// TIA Portal project "FB_zad2" (V15.1)

(* hardware
DEVICE "S7-1200 station_1"  S7-1200 Station
   slot 0: "Rack_0"  S7-1200 Rack  Rack  V1.0
   slot 1: "PLC_1"  CPU 1215C DC/DC/DC  6ES7 215-1AG40-0XB0  V4.2
*)

// ===== PLC "PLC_1"  CPU 1215C DC/DC/DC =====

VAR_GLOBAL   // PLC tag table "Default tag table"
   "OS1" AT %I1.0 : Bool;
   "OS2" AT %I0.7 : Bool;
   "P1" AT %Q1.0 : Bool;
   "P2" AT %Q0.7 : Bool;
   "P3_k_stolu" AT %Q0.5 : Bool;
   "P3_k_dopravniku" AT %Q0.6 : Bool;
   "P1_pracuje" AT %M10.0 : Bool;
   "P2_pracuje" AT %M10.1 : Bool;
   "P3_pracuje" AT %M10.2 : Bool;
   "Rotating_Table" AT %Q0.4 : Bool;
   "KS1" AT %I0.3 : Bool;
   "KS2" AT %I0.6 : Bool;
   "Table_Is_Ok" AT %M10.3 : Bool;
   "D1" AT %Q0.2 : Bool;
   "OS3" AT %I0.2 : Bool;
   "kompressor" AT %Q0.0 : Bool;
   "poz2_pom" AT %M10.4 : Bool;
END_VAR

DATA_BLOCK "P1_DB"   // DB1
{ S7_Optimized_Access := 'TRUE' }
VERSION : 0.1
// stored: InstanceOfName Piston_FB
"Piston_FB"
BEGIN
   i_Sensor_Low := true;
   i_Sensor_High := true;
END_DATA_BLOCK

DATA_BLOCK "P2_DB"   // DB2
{ S7_Optimized_Access := 'TRUE' }
VERSION : 0.1
// stored: InstanceOfName Piston_FB
"Piston_FB"
BEGIN
END_DATA_BLOCK

DATA_BLOCK "P3_DB"   // DB3
{ S7_Optimized_Access := 'TRUE' }
VERSION : 0.1
// stored: InstanceOfName Piston_FB
"Piston_FB"
BEGIN
   i_Is_Big_Piston := true;
END_DATA_BLOCK

DATA_BLOCK "Table1_DB"   // DB4
{ S7_Optimized_Access := 'TRUE' }
VERSION : 0.1
// stored: InstanceOfName Rotating_Table_FB
"Rotating_Table_FB"
BEGIN
END_DATA_BLOCK

DATA_BLOCK "Conv_DB"   // DB5
{ S7_Optimized_Access := 'TRUE' }
VERSION : 0.1
// stored: InstanceOfName Conveyor_FB
"Conveyor_FB"
BEGIN
END_DATA_BLOCK

FUNCTION_BLOCK "Piston_FB"   // FB1, LAD
{ S7_Optimized_Access := 'TRUE' }
VERSION : 0.1
   VAR_INPUT
      i_Enable : Bool;   // Personal control
      i_Is_Big_Piston : Bool;   // (поршни с двумя outputs, то есть как Р3)
      i_Use_Sensors : Bool;   // (true only for P1)
      i_Sensor_Low : Bool;   // (OS1)
      i_Sensor_High : Bool;   // (OS2)
      i_Set_Count : Int;   // (N iterations)
   END_VAR
   VAR_OUTPUT
      q_Forward : Bool;   // (k stolu)
      q_Backward : Bool;   // (od stola)
      q_Done : Bool;   // (Don't work)
      q_Busy : Bool;   // (In process)
      q_Object_ID : Int;
   END_VAR
   VAR
      Timer_For_Detection : TON_TIME;
      S_Vyska_Zistena : Bool;
      Timer_Work : TON_TIME;
      Timer_Return : TON_TIME;
      s_Counter_Val : Int;
      s_Edge_Mem : Bool;
      Timer_To_Push : TON_TIME;
   END_VAR
   VAR_TEMP   // added for the SCL form of the ladder/FBD networks
      _w1 : Bool;
   END_VAR
BEGIN

REGION Network 1: Určenie výšky objektu (funguje len pre prvý piest)
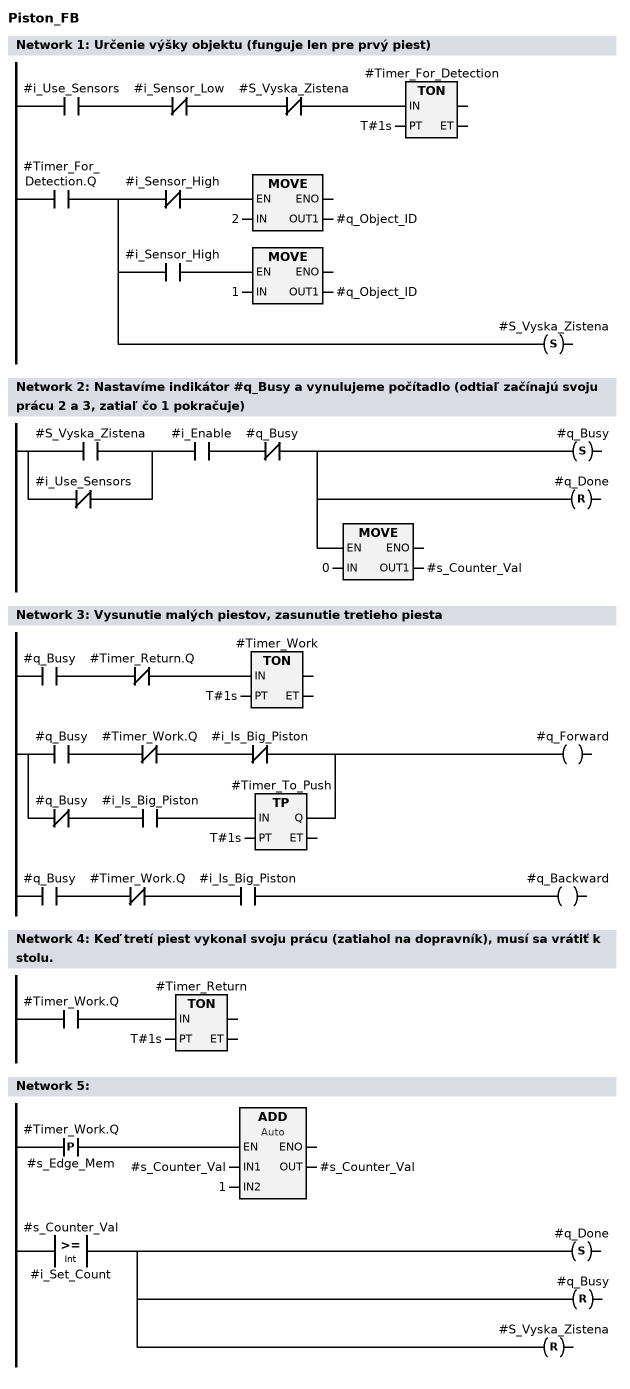
   #Timer_For_Detection(IN := #i_Use_Sensors AND NOT #i_Sensor_Low AND NOT #S_Vyska_Zistena, PT := T#1s);   // TON
   IF #Timer_For_Detection.Q AND NOT #i_Sensor_High THEN #q_Object_ID := 2; END_IF;
   IF #Timer_For_Detection.Q AND #i_Sensor_High THEN #q_Object_ID := 1; END_IF;
   IF #Timer_For_Detection.Q THEN #S_Vyska_Zistena := TRUE; END_IF;
END_REGION

REGION Network 2: Nastavíme indikátor #q_Busy a vynulujeme počítadlo (odtiaľ začínajú svoju prácu 2 a 3, zatiaľ čo 1 pokračuje)
   RUNG wire#powerrail
      Contact( #S_Vyska_Zistena )
      wire#w1
      Contact( #i_Enable )
      I_Contact( #q_Busy )
      wire#w2
      S_Coil( #q_Busy )
   END_RUNG
   RUNG wire#powerrail
      I_Contact( #i_Use_Sensors )
   END_RUNG wire#w1
   RUNG wire#w2
      R_Coil( #q_Done )
   END_RUNG
   RUNG wire#w2
      Move(in := 0, out1 => #s_Counter_Val)
   END_RUNG
   // the same network as SCL:
   #_w1 := (#S_Vyska_Zistena OR NOT #i_Use_Sensors) AND #i_Enable AND NOT #q_Busy;
   IF #_w1 THEN
       #q_Busy := TRUE;
       #q_Done := FALSE;
       #s_Counter_Val := 0;
   END_IF;
END_REGION

REGION Network 3: Vysunutie malých piestov, zasunutie tretieho piesta
   #Timer_Work(IN := #q_Busy AND NOT #Timer_Return.Q, PT := T#1s);   // TON
   #Timer_To_Push(IN := NOT #q_Busy AND #i_Is_Big_Piston, PT := T#1s);   // TP
   #q_Forward := (#q_Busy AND NOT #Timer_Work.Q AND NOT #i_Is_Big_Piston) OR #Timer_To_Push.Q;
   #q_Backward := #q_Busy AND NOT #Timer_Work.Q AND #i_Is_Big_Piston;
END_REGION

REGION Network 4: Keď tretí piest vykonal svoju prácu (zatiahol na dopravník), musí sa vrátiť k stolu.
   #Timer_Return(IN := #Timer_Work.Q, PT := T#1s);   // TON
END_REGION

REGION Network 5
   RUNG wire#powerrail
      P_Contact(operand := #Timer_Work.Q, bit := #s_Edge_Mem)
      Add(in1 := #s_Counter_Val, in2 := 1, out => #s_Counter_Val)
   END_RUNG
   RUNG wire#powerrail
      { S7_Templates := "SrcType := Int" } GE_Contact(in1 := #s_Counter_Val, in2 := #i_Set_Count)
      wire#w1
      S_Coil( #q_Done )
   END_RUNG
   RUNG wire#w1
      R_Coil( #q_Busy )
   END_RUNG
   RUNG wire#w1
      R_Coil( #S_Vyska_Zistena )
   END_RUNG
   // the same network as SCL:
   #_w1 := #Timer_Work.Q AND NOT #s_Edge_Mem;   // rising edge of #Timer_Work.Q
   #s_Edge_Mem := #Timer_Work.Q;
   IF #_w1 THEN #s_Counter_Val := #s_Counter_Val + 1; END_IF;
   IF #s_Counter_Val >= #i_Set_Count THEN
       #q_Done := TRUE;
       #q_Busy := FALSE;
       #S_Vyska_Zistena := FALSE;
   END_IF;
END_REGION
END_FUNCTION_BLOCK

FUNCTION_BLOCK "Rotating_Table_FB"   // FB2, LAD
{ S7_Optimized_Access := 'TRUE' }
VERSION : 0.1
   VAR_INPUT
      i_Enable_Auto : Bool;
      i_Enable_Manual : Bool;   // KS1
      i_Loading : Bool;   // Signal "Done" from P1_DB
      i_New_ID : Int;   // ID from P1_DB for poz1
      i_Confirm_Button : Bool;   // KS2
      i_Unloading : Bool;
   END_VAR
   VAR_OUTPUT
      q_State_Ok : Bool;
      q_Motor : Bool;
      q_Start_Poz_State : Bool;
   END_VAR
   VAR
      s_Poz1 : Int;
      s_poz2_id : Bool;
      s_Poz2 : Int;
      s_Poz3 : Int;
      s_Poz4 : Int;
      s_Block_Rotation : Bool;
      s_Need_Rotation : Bool;
      s_Rotation_Time : TON_TIME;
      s_Loading_Pom : Bool;
      s_Timer_Rotation_Pom : Bool;
      s_Timer_Rotation_Pom2 : Bool;
      s_Unloading_Pom : Bool;
      s_Rotation_Time2 : TON_TIME;
   END_VAR
   VAR_TEMP   // added for the SCL form of the ladder/FBD networks
      _w1 : Bool;
      _w2 : Bool;
   END_VAR
BEGIN

REGION Network 1
   // Vynulovanie poz3
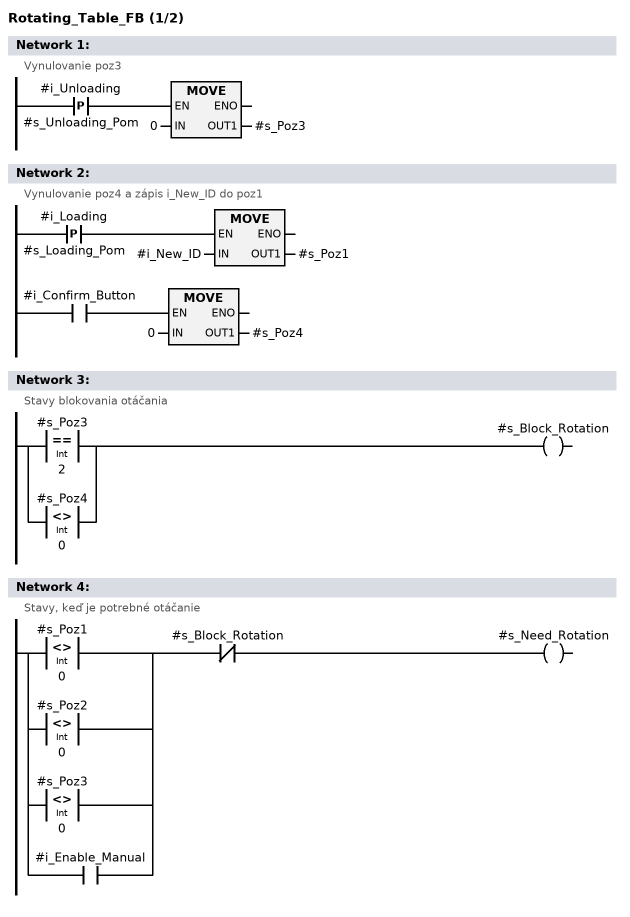
   RUNG wire#powerrail
      P_Contact(operand := #i_Unloading, bit := #s_Unloading_Pom)
      Move(in := 0, out1 => #s_Poz3)
   END_RUNG
   // the same network as SCL:
   #_w1 := #i_Unloading AND NOT #s_Unloading_Pom;   // rising edge of #i_Unloading
   #s_Unloading_Pom := #i_Unloading;
   IF #_w1 THEN #s_Poz3 := 0; END_IF;
END_REGION

REGION Network 2
   // Vynulovanie poz4 a zápis i_New_ID do poz1
   RUNG wire#powerrail
      P_Contact(operand := #i_Loading, bit := #s_Loading_Pom)
      Move(in := #i_New_ID, out1 => #s_Poz1)
   END_RUNG
   RUNG wire#powerrail
      Contact( #i_Confirm_Button )
      Move(in := 0, out1 => #s_Poz4)
   END_RUNG
   // the same network as SCL:
   #_w1 := #i_Loading AND NOT #s_Loading_Pom;   // rising edge of #i_Loading
   #s_Loading_Pom := #i_Loading;
   IF #_w1 THEN #s_Poz1 := #i_New_ID; END_IF;
   IF #i_Confirm_Button THEN #s_Poz4 := 0; END_IF;
END_REGION

REGION Network 3
   // Stavy blokovania otáčania
   RUNG wire#powerrail
      { S7_Templates := "SrcType := Int" } EQ_Contact(in1 := #s_Poz3, in2 := 2)
      wire#w1
      Coil( #s_Block_Rotation )
   END_RUNG
   RUNG wire#powerrail
      { S7_Templates := "SrcType := Int" } NE_Contact(in1 := #s_Poz4, in2 := 0)
   END_RUNG wire#w1
   // the same network as SCL:
   #s_Block_Rotation := (#s_Poz3 = 2) OR (#s_Poz4 <> 0);
END_REGION

REGION Network 4
   // Stavy, keď je potrebné otáčanie
   RUNG wire#powerrail
      { S7_Templates := "SrcType := Int" } NE_Contact(in1 := #s_Poz1, in2 := 0)
      wire#w1
      I_Contact( #s_Block_Rotation )
      Coil( #s_Need_Rotation )
   END_RUNG
   RUNG wire#powerrail
      { S7_Templates := "SrcType := Int" } NE_Contact(in1 := #s_Poz2, in2 := 0)
   END_RUNG wire#w1
   RUNG wire#powerrail
      { S7_Templates := "SrcType := Int" } NE_Contact(in1 := #s_Poz3, in2 := 0)
   END_RUNG wire#w1
   RUNG wire#powerrail
      Contact( #i_Enable_Manual )
   END_RUNG wire#w1
   // the same network as SCL:
   #s_Need_Rotation := ((#s_Poz1 <> 0) OR (#s_Poz2 <> 0) OR (#s_Poz3 <> 0) OR #i_Enable_Manual) AND NOT #s_Block_Rotation;
END_REGION

REGION Network 5
   // Určite pridanie druhého časovača (TR) nie je najstručnejším riešením, ale funguje to :))
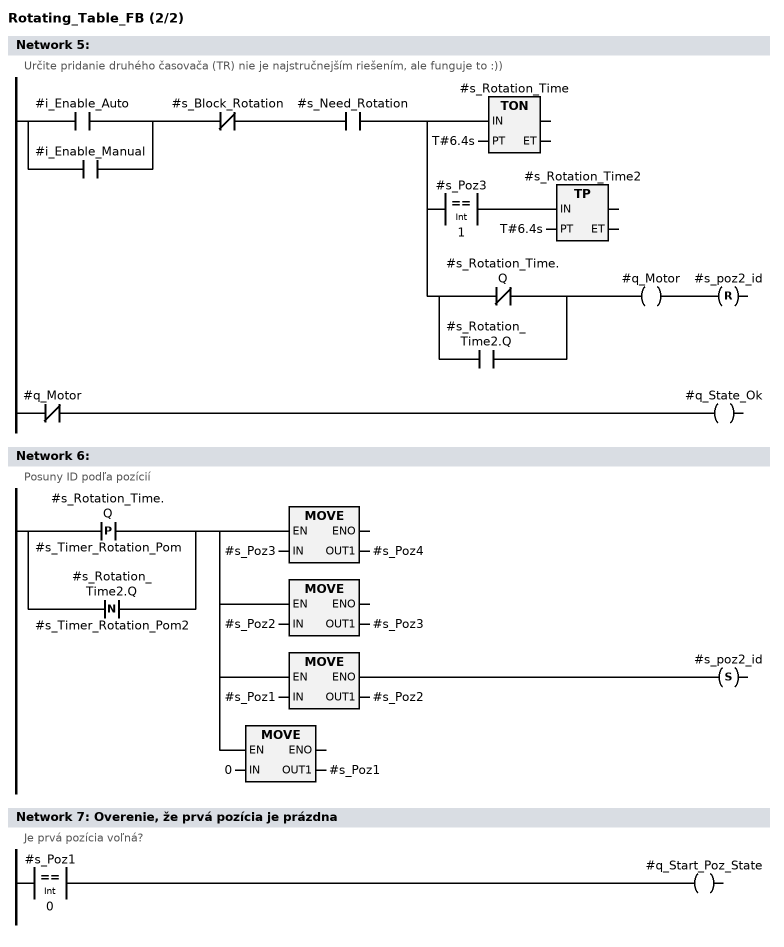
   #_w1 := (#i_Enable_Auto OR #i_Enable_Manual) AND NOT #s_Block_Rotation AND #s_Need_Rotation;
   #s_Rotation_Time(IN := #_w1, PT := T#6.4s);   // TON
   #s_Rotation_Time2(IN := #_w1 AND (#s_Poz3 = 1), PT := T#6.4s);   // TP
   #q_Motor := #_w1 AND (NOT #s_Rotation_Time.Q OR #s_Rotation_Time2.Q);
   IF #q_Motor THEN #s_poz2_id := FALSE; END_IF;
   #q_State_Ok := NOT #q_Motor;
END_REGION

REGION Network 6
   // Posuny ID podľa pozícií
   RUNG wire#powerrail
      P_Contact(operand := #s_Rotation_Time.Q, bit := #s_Timer_Rotation_Pom)
      wire#w1
      Move(in := #s_Poz3, out1 => #s_Poz4)
   END_RUNG
   RUNG wire#powerrail
      N_Contact(operand := #s_Rotation_Time2.Q, bit := #s_Timer_Rotation_Pom2)
   END_RUNG wire#w1
   RUNG wire#w1
      Move(in := #s_Poz2, out1 => #s_Poz3)
   END_RUNG
   RUNG wire#w1
      Move(in := #s_Poz1, out1 => #s_Poz2)
      S_Coil( #s_poz2_id )
   END_RUNG
   RUNG wire#w1
      Move(in := 0, out1 => #s_Poz1)
   END_RUNG
   // the same network as SCL:
   #_w1 := #s_Rotation_Time.Q AND NOT #s_Timer_Rotation_Pom;   // rising edge of #s_Rotation_Time.Q
   #s_Timer_Rotation_Pom := #s_Rotation_Time.Q;
   #_w2 := NOT #s_Rotation_Time2.Q AND #s_Timer_Rotation_Pom2;   // falling edge of #s_Rotation_Time2.Q
   #s_Timer_Rotation_Pom2 := #s_Rotation_Time2.Q;
   IF #_w1 OR #_w2 THEN
       #s_Poz4 := #s_Poz3;
       #s_Poz3 := #s_Poz2;
       #s_Poz2 := #s_Poz1;
       #s_poz2_id := TRUE;
       #s_Poz1 := 0;
   END_IF;
END_REGION

REGION Network 7: Overenie, že prvá pozícia je prázdna
   // Je prvá pozícia voľná?
   RUNG wire#powerrail
      { S7_Templates := "SrcType := Int" } EQ_Contact(in1 := #s_Poz1, in2 := 0)
      Coil( #q_Start_Poz_State )
   END_RUNG
   // the same network as SCL:
   #q_Start_Poz_State := #s_Poz1 = 0;
END_REGION
END_FUNCTION_BLOCK

FUNCTION_BLOCK "Conveyor_FB"   // FB4, LAD
{ S7_Optimized_Access := 'TRUE' }
VERSION : 0.1
   VAR_INPUT
      i_Sensor : Bool;
      i_Loading : Bool;   // Signal P3.Done
      i_New_ID : Int;
   END_VAR
   VAR_OUTPUT
      q_Motor : Bool;
      q_Entry_Is_Free : Bool;
   END_VAR
   VAR
      s_Poz5 : Int;
      s_Poz6 : Int;
      s_Is_poz6_Free : Bool;
      s_Sensor_Fall : Bool;
      s_Sensor_Rise : Bool;
      s_Loading_Pom : Bool;
   END_VAR
   VAR_TEMP   // added for the SCL form of the ladder/FBD networks
      _w1 : Bool;
   END_VAR
BEGIN

REGION Network 1: Keď piest pretiahol objekt, zapíš ID do piatej pozície
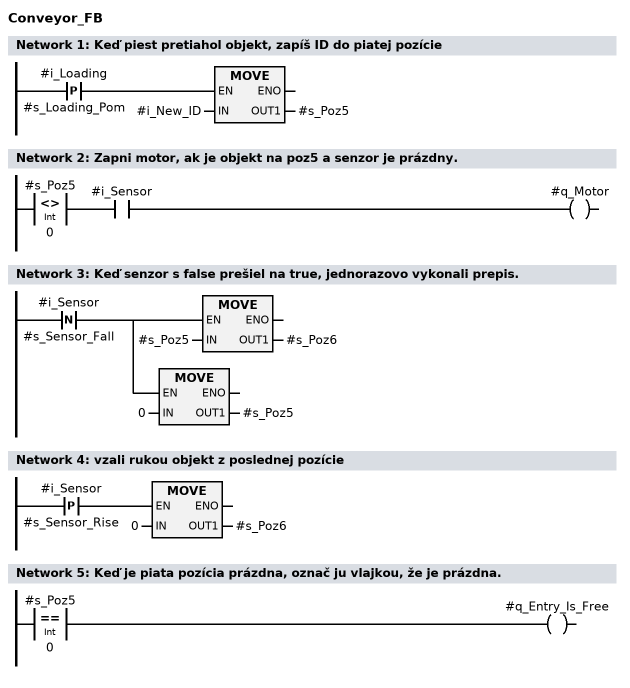
   RUNG wire#powerrail
      P_Contact(operand := #i_Loading, bit := #s_Loading_Pom)
      Move(in := #i_New_ID, out1 => #s_Poz5)
   END_RUNG
   // the same network as SCL:
   #_w1 := #i_Loading AND NOT #s_Loading_Pom;   // rising edge of #i_Loading
   #s_Loading_Pom := #i_Loading;
   IF #_w1 THEN #s_Poz5 := #i_New_ID; END_IF;
END_REGION

REGION Network 2: Zapni motor, ak je objekt na poz5 a senzor je prázdny.
   RUNG wire#powerrail
      { S7_Templates := "SrcType := Int" } NE_Contact(in1 := #s_Poz5, in2 := 0)
      Contact( #i_Sensor )
      Coil( #q_Motor )
   END_RUNG
   // the same network as SCL:
   #q_Motor := (#s_Poz5 <> 0) AND #i_Sensor;
END_REGION

REGION Network 3: Keď senzor s false prešiel na true, jednorazovo vykonali prepis.
   RUNG wire#powerrail
      N_Contact(operand := #i_Sensor, bit := #s_Sensor_Fall)
      wire#w1
      Move(in := #s_Poz5, out1 => #s_Poz6)
   END_RUNG
   RUNG wire#w1
      Move(in := 0, out1 => #s_Poz5)
   END_RUNG
   // the same network as SCL:
   #_w1 := NOT #i_Sensor AND #s_Sensor_Fall;   // falling edge of #i_Sensor
   #s_Sensor_Fall := #i_Sensor;
   IF #_w1 THEN
       #s_Poz6 := #s_Poz5;
       #s_Poz5 := 0;
   END_IF;
END_REGION

REGION Network 4: vzali rukou objekt z poslednej pozície
   RUNG wire#powerrail
      P_Contact(operand := #i_Sensor, bit := #s_Sensor_Rise)
      Move(in := 0, out1 => #s_Poz6)
   END_RUNG
   // the same network as SCL:
   #_w1 := #i_Sensor AND NOT #s_Sensor_Rise;   // rising edge of #i_Sensor
   #s_Sensor_Rise := #i_Sensor;
   IF #_w1 THEN #s_Poz6 := 0; END_IF;
END_REGION

REGION Network 5: Keď je piata pozícia prázdna, označ ju vlajkou, že je prázdna.
   RUNG wire#powerrail
      { S7_Templates := "SrcType := Int" } EQ_Contact(in1 := #s_Poz5, in2 := 0)
      Coil( #q_Entry_Is_Free )
   END_RUNG
   // the same network as SCL:
   #q_Entry_Is_Free := #s_Poz5 = 0;
END_REGION
END_FUNCTION_BLOCK

ORGANIZATION_BLOCK "Main"   // OB1, LAD, ProgramCycle
TITLE = "Main Program Sweep (Cycle)"
{ S7_Optimized_Access := 'TRUE' }
VERSION : 0.1
   VAR_INPUT
      Initial_Call : Bool;   // Initial call of this OB
      Remanence : Bool;   // =True, if remanent data are available
   END_VAR
   VAR_TEMP   // added for the SCL form of the ladder/FBD networks
      _w1 : Bool;
   END_VAR
BEGIN

REGION Network 1: Je mozno dat ( ) namiesto Set
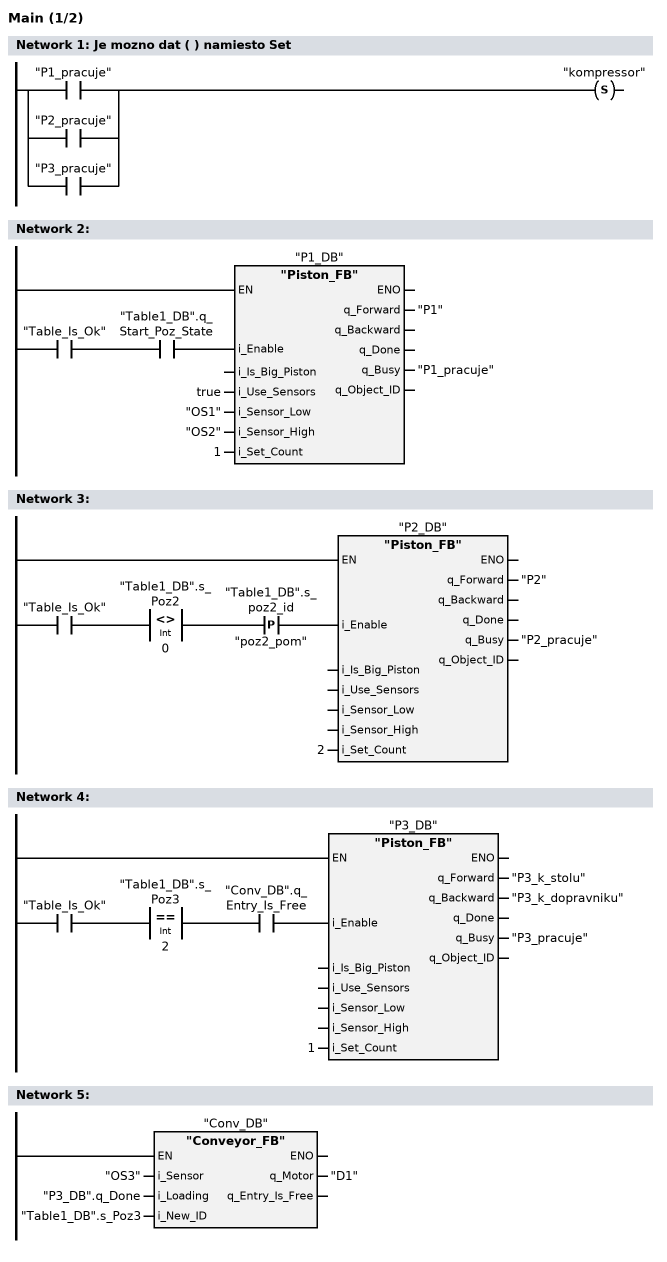
   RUNG wire#powerrail
      Contact( "P1_pracuje" )
      wire#w1
      S_Coil( "kompressor" )
   END_RUNG
   RUNG wire#powerrail
      Contact( "P2_pracuje" )
   END_RUNG wire#w1
   RUNG wire#powerrail
      Contact( "P3_pracuje" )
   END_RUNG wire#w1
   // the same network as SCL:
   IF "P1_pracuje" OR "P2_pracuje" OR "P3_pracuje" THEN "kompressor" := TRUE; END_IF;
END_REGION

REGION Network 2
   RUNG wire#powerrail
      "P1_DB"(i_Enable := wire#w1, i_Is_Big_Piston :=, i_Use_Sensors := true, i_Sensor_Low := "OS1", i_Sensor_High := "OS2", i_Set_Count := 1, q_Forward => "P1", q_Backward =>, q_Done =>, q_Busy => "P1_pracuje", q_Object_ID =>)
   END_RUNG
   RUNG wire#powerrail
      Contact( "Table_Is_Ok" )
      Contact( "Table1_DB".q_Start_Poz_State )
   END_RUNG wire#w1
   // the same network as SCL:
   "P1_DB"(i_Enable := "Table_Is_Ok" AND "Table1_DB".q_Start_Poz_State,   // "Piston_FB"
           i_Use_Sensors := true,
           i_Sensor_Low := "OS1",
           i_Sensor_High := "OS2",
           i_Set_Count := 1,
           q_Forward => "P1",
           q_Busy => "P1_pracuje");
END_REGION

REGION Network 3
   RUNG wire#powerrail
      "P2_DB"(i_Enable := wire#w1, i_Is_Big_Piston :=, i_Use_Sensors :=, i_Sensor_Low :=, i_Sensor_High :=, i_Set_Count := 2, q_Forward => "P2", q_Backward =>, q_Done =>, q_Busy => "P2_pracuje", q_Object_ID =>)
   END_RUNG
   RUNG wire#powerrail
      Contact( "Table_Is_Ok" )
      { S7_Templates := "SrcType := Int" } NE_Contact(in1 := "Table1_DB".s_Poz2, in2 := 0)
      P_Contact(operand := "Table1_DB".s_poz2_id, bit := "poz2_pom")
   END_RUNG wire#w1
   // the same network as SCL:
   #_w1 := "Table_Is_Ok" AND ("Table1_DB".s_Poz2 <> 0) AND "Table1_DB".s_poz2_id AND NOT "poz2_pom";   // rising edge of "Table1_DB".s_poz2_id
   "poz2_pom" := "Table1_DB".s_poz2_id;
   "P2_DB"(i_Enable := #_w1, i_Set_Count := 2, q_Forward => "P2", q_Busy => "P2_pracuje");   // "Piston_FB"
END_REGION

REGION Network 4
   RUNG wire#powerrail
      "P3_DB"(i_Enable := wire#w1, i_Is_Big_Piston :=, i_Use_Sensors :=, i_Sensor_Low :=, i_Sensor_High :=, i_Set_Count := 1, q_Forward => "P3_k_stolu", q_Backward => "P3_k_dopravniku", q_Done =>, q_Busy => "P3_pracuje", q_Object_ID =>)
   END_RUNG
   RUNG wire#powerrail
      Contact( "Table_Is_Ok" )
      { S7_Templates := "SrcType := Int" } EQ_Contact(in1 := "Table1_DB".s_Poz3, in2 := 2)
      Contact( "Conv_DB".q_Entry_Is_Free )
   END_RUNG wire#w1
   // the same network as SCL:
   "P3_DB"(i_Enable := "Table_Is_Ok" AND ("Table1_DB".s_Poz3 = 2) AND "Conv_DB".q_Entry_Is_Free,   // "Piston_FB"
           i_Set_Count := 1,
           q_Forward => "P3_k_stolu",
           q_Backward => "P3_k_dopravniku",
           q_Busy => "P3_pracuje");
END_REGION

REGION Network 5
   RUNG wire#powerrail
      "Conv_DB"(i_Sensor := "OS3", i_Loading := "P3_DB".q_Done, i_New_ID := "Table1_DB".s_Poz3, q_Motor => "D1", q_Entry_Is_Free =>)
   END_RUNG
   // the same network as SCL:
   "Conv_DB"(i_Sensor := "OS3", i_Loading := "P3_DB".q_Done, i_New_ID := "Table1_DB".s_Poz3, q_Motor => "D1");   // "Conveyor_FB"
END_REGION

REGION Network 6
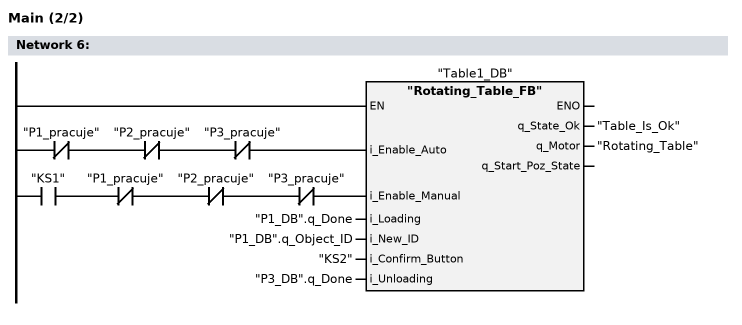
   RUNG wire#powerrail
      "Table1_DB"(i_Enable_Auto := wire#w1, i_Enable_Manual := wire#w2, i_Loading := "P1_DB".q_Done, i_New_ID := "P1_DB".q_Object_ID, i_Confirm_Button := "KS2", i_Unloading := "P3_DB".q_Done, q_State_Ok => "Table_Is_Ok", q_Motor => "Rotating_Table", q_Start_Poz_State =>)
   END_RUNG
   RUNG wire#powerrail
      I_Contact( "P1_pracuje" )
      I_Contact( "P2_pracuje" )
      I_Contact( "P3_pracuje" )
   END_RUNG wire#w1
   RUNG wire#powerrail
      Contact( "KS1" )
      I_Contact( "P1_pracuje" )
      I_Contact( "P2_pracuje" )
      I_Contact( "P3_pracuje" )
   END_RUNG wire#w2
   // the same network as SCL:
   "Table1_DB"(i_Enable_Auto := NOT "P1_pracuje" AND NOT "P2_pracuje" AND NOT "P3_pracuje",   // "Rotating_Table_FB"
               i_Enable_Manual := "KS1" AND NOT "P1_pracuje" AND NOT "P2_pracuje" AND NOT "P3_pracuje",
               i_Loading := "P1_DB".q_Done,
               i_New_ID := "P1_DB".q_Object_ID,
               i_Confirm_Button := "KS2",
               i_Unloading := "P3_DB".q_Done,
               q_State_Ok => "Table_Is_Ok",
               q_Motor => "Rotating_Table");
END_REGION
END_ORGANIZATION_BLOCK